FUNCTION_BLOCK FB_counter
VAR_INPUT
	iCounterStep : INT := 1;
END_VAR
VAR_OUTPUT
	iCounterOut : INT;
END_VAR
VAR
	iCounter : INT := 0;
END_VAR

iCounter := iCounter + iCounterStep;

END_FUNCTION_BLOCK

(* stored: Version 1.1.0.1, ProductVersion 3.1.4024.9
   POU FB_counter: Id {0dcfbd8b-c291-48eb-b185-90020c8b62bd}, SpecialFunc None *)
